PROGRAM S1_01_Motion_2
VAR
	HMI_Motion: FB_HMI_Control;
	Motion: FB_Motion2way;

	tMessageOffset: UINT;
	tNumMessagesPerRow: UINT;
	
	
	MyAdvanceInterlock: BOOL;
	MyReturnInterlock: BOOL;
	
	MyAutoAdvanceCondition: BOOL;
	MyAutoReturnCondition: BOOL;
	testword: WORD;
	myAdvancePrompt: BOOL;
	myReturnPrompt: BOOL;
	advancedSensor: BOOL;
	returnedSensor: BOOL;
	AdvanceCoil: BOOL;
	ReturnCoil: BOOL;
	tWaitMsgXICAdv: BOOL;
	tWaitMsgXICRet: BOOL;
	FB_SimMotion: FB_SimMotion;
END_VAR

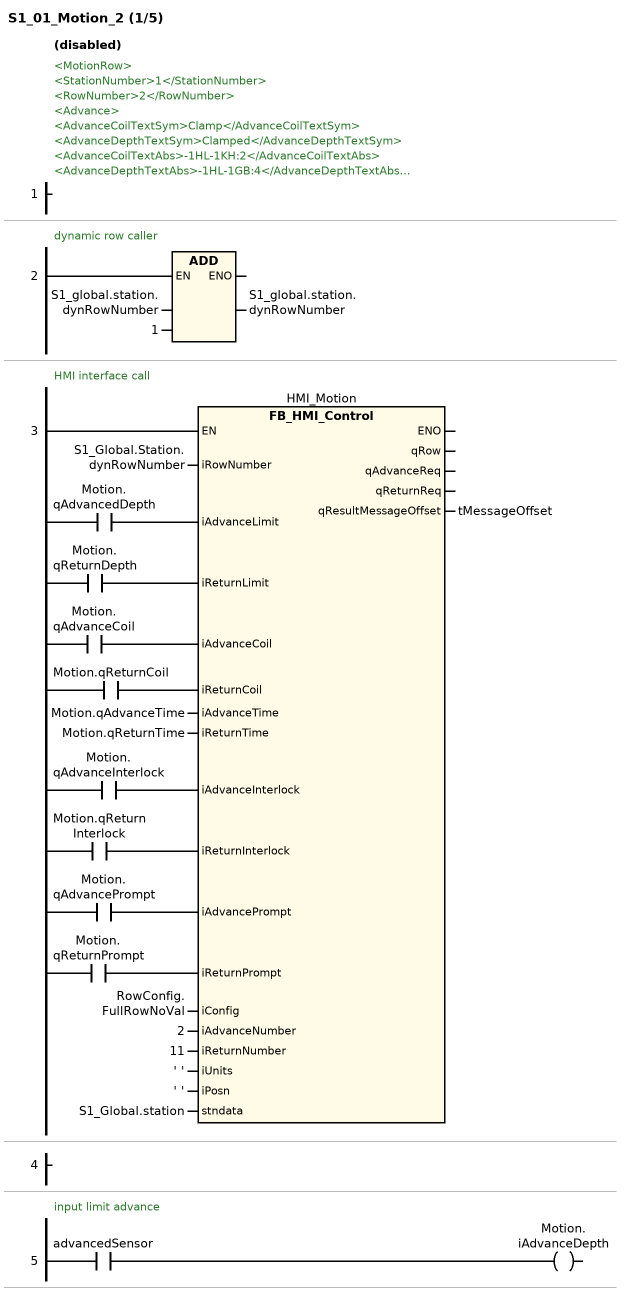
// NETWORK 1 (disabled)
// <MotionRow>
// <StationNumber>1</StationNumber>
// <RowNumber>2</RowNumber>
//   <Advance>
//     <AdvanceCoilTextSym>Clamp</AdvanceCoilTextSym>
//     <AdvanceDepthTextSym>Clamped</AdvanceDepthTextSym>
//     <AdvanceCoilTextAbs>-1HL-1KH:2</AdvanceCoilTextAbs>
//     <AdvanceDepthTextAbs>-1HL-1GB:4</AdvanceDepthTextAbs>
//     <ManSeq>2</ManSeq>
//   </Advance>
//   <Return>
//     <ReturnCoilTextSym>Unclamp</ReturnCoilTextSym>
//     <ReturnDepthTextSym>Unclamped</ReturnDepthTextSym>
//     <ReturnCoilTextAbs>-1HL-1KH:4</ReturnCoilTextAbs>
//     <ReturnDepthTextAbs>-1HL-2BG:4</ReturnDepthTextAbs>
//    <ManSeq>11</ManSeq>
//   </Return>
//   <Motion>
//     <NameSym>Part Clamp 1</NameSym>
//     <NameAbs>-1HL-1UQ</NameAbs>
//   </Motion>
// </MotionRow>

// NETWORK 2
// dynamic row caller
S1_global.station.dynRowNumber := S1_global.station.dynRowNumber + 1;

// NETWORK 3
// HMI interface call
HMI_Motion(
    iRowNumber := S1_Global.Station.dynRowNumber,
    iAdvanceLimit := Motion.qAdvancedDepth,
    iReturnLimit := Motion.qReturnDepth,
    iAdvanceCoil := Motion.qAdvanceCoil,
    iReturnCoil := Motion.qReturnCoil,
    iAdvanceTime := Motion.qAdvanceTime,
    iReturnTime := Motion.qReturnTime,
    iAdvanceInterlock := Motion.qAdvanceInterlock,
    iReturnInterlock := Motion.qReturnInterlock,
    iAdvancePrompt := Motion.qAdvancePrompt,
    iReturnPrompt := Motion.qReturnPrompt,
    iConfig := RowConfig.FullRowNoVal,
    iAdvanceNumber := 2,
    iReturnNumber := 11,
    iUnits := ' ',
    iPosn := ' ',
    stndata := S1_Global.station,
    qResultMessageOffset => tMessageOffset); // FB_HMI_Control

// NETWORK 4

// NETWORK 5
// input limit advance
Motion.iAdvanceDepth := advancedSensor;

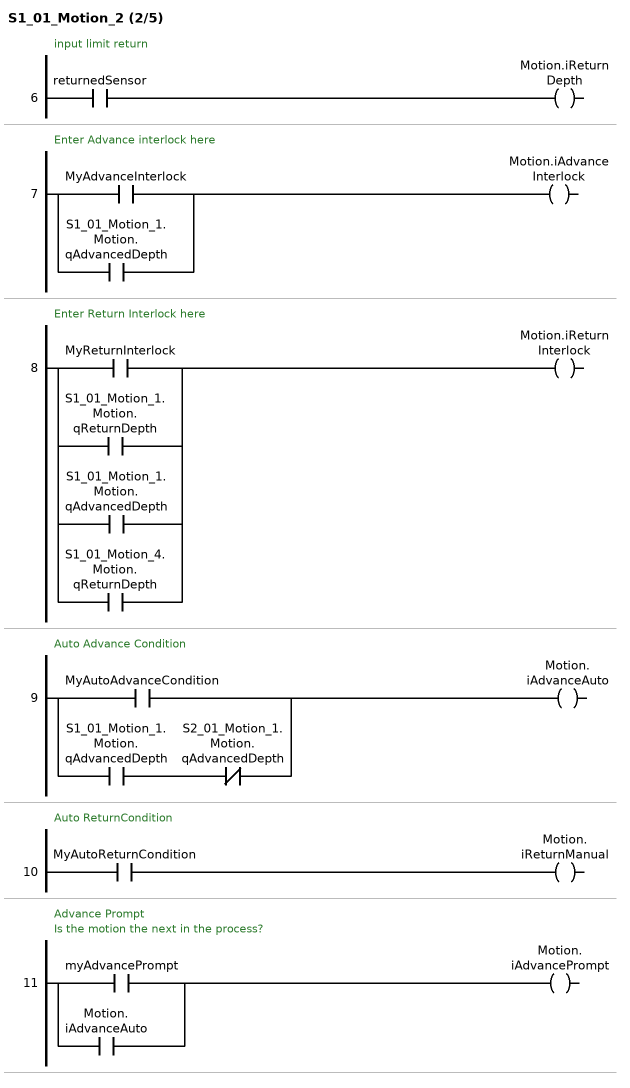
// NETWORK 6
// input limit return
Motion.iReturnDepth := returnedSensor;

// NETWORK 7
// Enter Advance interlock here
Motion.iAdvanceInterlock := MyAdvanceInterlock OR S1_01_Motion_1.Motion.qAdvancedDepth;

// NETWORK 8
// Enter Return Interlock here
Motion.iReturnInterlock := MyReturnInterlock OR S1_01_Motion_1.Motion.qReturnDepth OR S1_01_Motion_1.Motion.qAdvancedDepth OR S1_01_Motion_4.Motion.qReturnDepth;

// NETWORK 9
// Auto Advance Condition
Motion.iAdvanceAuto := MyAutoAdvanceCondition OR S1_01_Motion_1.Motion.qAdvancedDepth AND NOT S2_01_Motion_1.Motion.qAdvancedDepth;

// NETWORK 10
// Auto ReturnCondition
Motion.iReturnManual := MyAutoReturnCondition;

// NETWORK 11
// Advance Prompt
// Is the motion the next in the process?
Motion.iAdvancePrompt := myAdvancePrompt OR Motion.iAdvanceAuto;

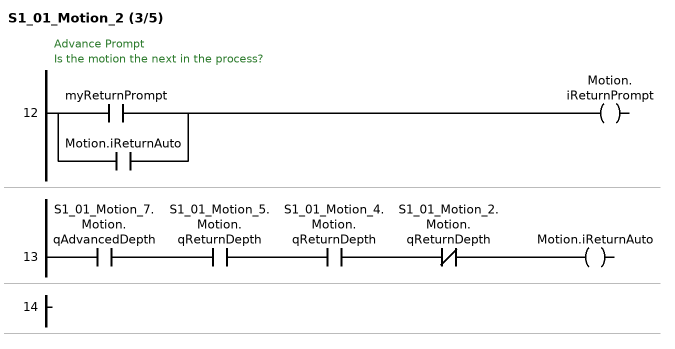
// NETWORK 12
// Advance Prompt
// Is the motion the next in the process?
Motion.iReturnPrompt := myReturnPrompt OR Motion.iReturnAuto;

// NETWORK 13
Motion.iReturnAuto := S1_01_Motion_7.Motion.qAdvancedDepth AND S1_01_Motion_5.Motion.qReturnDepth AND S1_01_Motion_4.Motion.qReturnDepth AND NOT S1_01_Motion_2.Motion.qReturnDepth;

// NETWORK 14

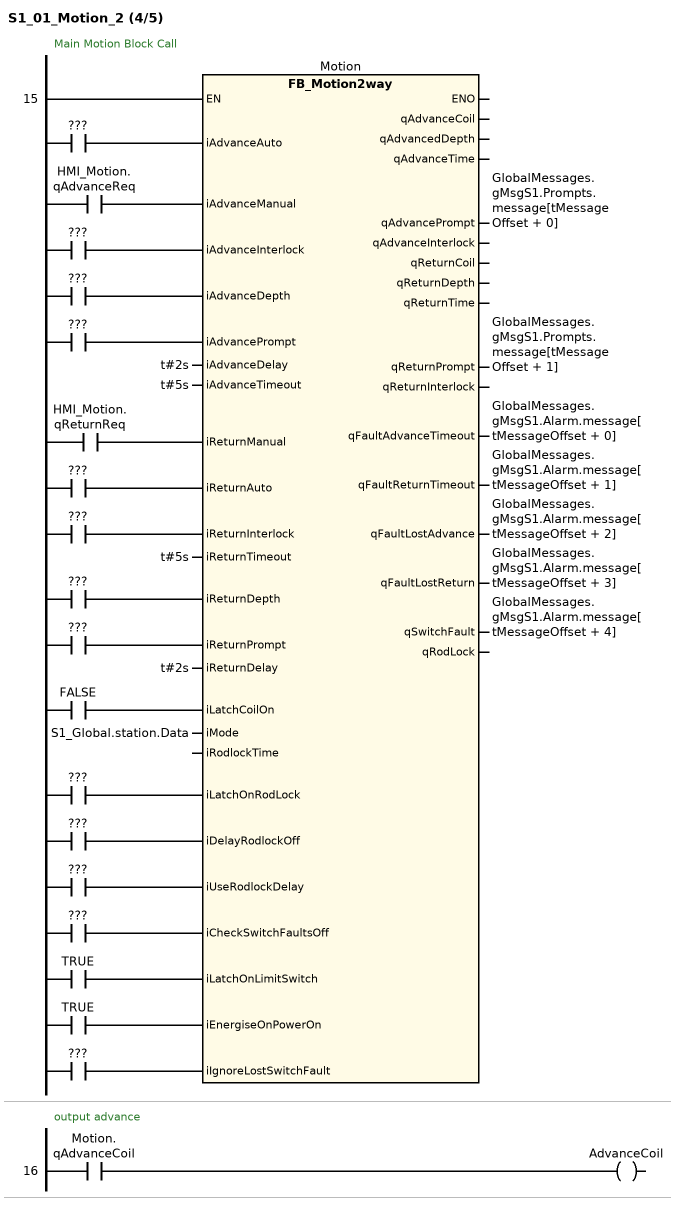
// NETWORK 15
// Main Motion Block Call
Motion(
    iAdvanceManual := HMI_Motion.qAdvanceReq,
    iAdvanceDelay := t#2s,
    iAdvanceTimeout := t#5s,
    iReturnManual := HMI_Motion.qReturnReq,
    iReturnTimeout := t#5s,
    iReturnDelay := t#2s,
    iLatchCoilOn := FALSE,
    iMode := S1_Global.station.Data,
    iLatchOnLimitSwitch := TRUE,
    iEnergiseOnPowerOn := TRUE,
    qAdvancePrompt => GlobalMessages.gMsgS1.Prompts.message[tMessageOffset + 0],
    qReturnPrompt => GlobalMessages.gMsgS1.Prompts.message[tMessageOffset + 1],
    qFaultAdvanceTimeout => GlobalMessages.gMsgS1.Alarm.message[tMessageOffset + 0],
    qFaultReturnTimeout => GlobalMessages.gMsgS1.Alarm.message[tMessageOffset + 1],
    qFaultLostAdvance => GlobalMessages.gMsgS1.Alarm.message[tMessageOffset + 2],
    qFaultLostReturn => GlobalMessages.gMsgS1.Alarm.message[tMessageOffset + 3],
    qSwitchFault => GlobalMessages.gMsgS1.Alarm.message[tMessageOffset + 4]); // FB_Motion2way

// NETWORK 16
// output advance
AdvanceCoil := Motion.qAdvanceCoil;

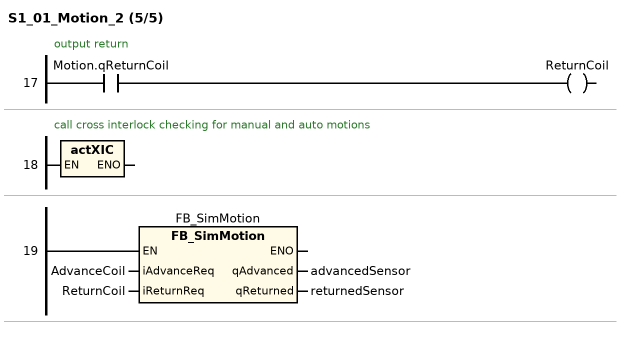
// NETWORK 17
// output return
ReturnCoil := Motion.qReturnCoil;

// NETWORK 18
// call cross interlock checking for manual and auto motions
actXIC();

// NETWORK 19
FB_SimMotion(
    iAdvanceReq := AdvanceCoil,
    iReturnReq := ReturnCoil,
    qAdvanced => advancedSensor,
    qReturned => returnedSensor);

ACTION actXIC:
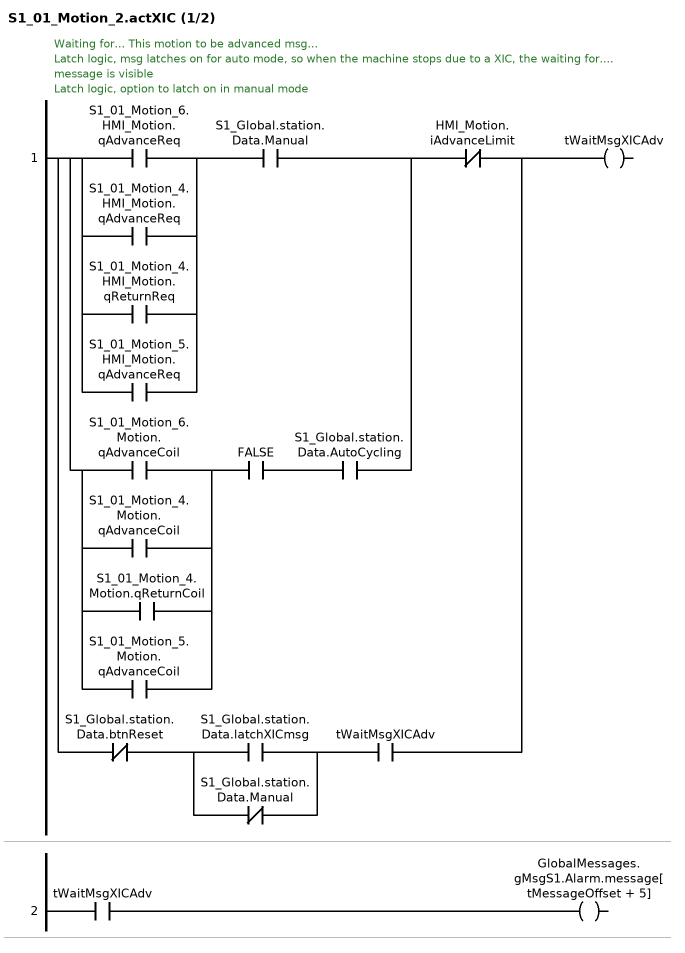
// NETWORK 1
// Waiting for... This motion to be advanced msg...
// Latch logic, msg latches on for auto mode, so when the machine stops due to a XIC, the waiting for.... message is visible
// Latch logic, option to latch on in manual mode
tWaitMsgXICAdv := ((S1_01_Motion_6.HMI_Motion.qAdvanceReq OR S1_01_Motion_4.HMI_Motion.qAdvanceReq OR S1_01_Motion_4.HMI_Motion.qReturnReq OR S1_01_Motion_5.HMI_Motion.qAdvanceReq) AND S1_Global.station.Data.Manual OR (S1_01_Motion_6.Motion.qAdvanceCoil OR S1_01_Motion_4.Motion.qAdvanceCoil OR S1_01_Motion_4.Motion.qReturnCoil OR S1_01_Motion_5.Motion.qAdvanceCoil) AND FALSE AND S1_Global.station.Data.AutoCycling) AND NOT HMI_Motion.iAdvanceLimit OR NOT S1_Global.station.Data.btnReset AND (S1_Global.station.Data.latchXICmsg OR NOT S1_Global.station.Data.Manual) AND tWaitMsgXICAdv;

// NETWORK 2
GlobalMessages.gMsgS1.Alarm.message[tMessageOffset + 5] := tWaitMsgXICAdv;

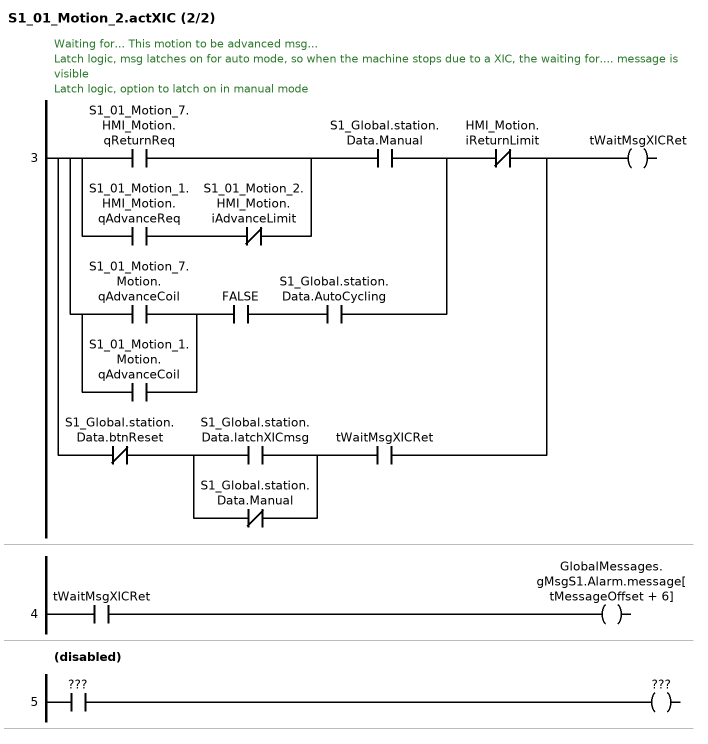
// NETWORK 3
// Waiting for... This motion to be advanced msg...
// Latch logic, msg latches on for auto mode, so when the machine stops due to a XIC, the waiting for.... message is visible
// Latch logic, option to latch on in manual mode
tWaitMsgXICRet := ((S1_01_Motion_7.HMI_Motion.qReturnReq OR S1_01_Motion_1.HMI_Motion.qAdvanceReq AND NOT S1_01_Motion_2.HMI_Motion.iAdvanceLimit) AND S1_Global.station.Data.Manual OR (S1_01_Motion_7.Motion.qAdvanceCoil OR S1_01_Motion_1.Motion.qAdvanceCoil) AND FALSE AND S1_Global.station.Data.AutoCycling) AND NOT HMI_Motion.iReturnLimit OR NOT S1_Global.station.Data.btnReset AND (S1_Global.station.Data.latchXICmsg OR NOT S1_Global.station.Data.Manual) AND tWaitMsgXICRet;

// NETWORK 4
GlobalMessages.gMsgS1.Alarm.message[tMessageOffset + 6] := tWaitMsgXICRet;

// NETWORK 5 (disabled)
// ??? := ???;
END_ACTION

END_PROGRAM

(* stored: Version 1.1.0.1, ProductVersion 3.1.4024.11
   POU S1_01_Motion_2: Id {10e806c2-25e2-4382-9a9a-c4fcfc43aa8b}, SpecialFunc None
   Action actXIC: Id {e00b4bd9-bf5a-0a4e-116e-cde3cd238250} *)
